FUNCTION_BLOCK CiA_DS402Controlword_Lenze EXTENDS CiA_DS402Controlword
VAR_INPUT
	ReleaseBrake			: BOOL; //Manufacturere specific Bit 14 
END_VAR
VAR_OUTPUT
END_VAR
VAR
END_VAR

;

METHOD PUBLIC createControlword : BOOL
VAR_INPUT
	StatusState												: eCiA_DS402_STATUS_STATE;
END_VAR
VAR_IN_OUT
	Controlword												:	UINT;
END_VAR
	
	createControlword											:= SUPER^.createControlword(StatusState,Controlword);;
	Controlword.14												:= ReleaseBrake;	
	
	

(*****************************************************************************)
END_METHOD

END_FUNCTION_BLOCK

(* stored: Version 1.1.0.1, ProductVersion 3.1.4024.13
   POU CiA_DS402Controlword_Lenze: Id {8f5f011b-553f-44e1-a91b-77b2decd4123}, SpecialFunc None
   Method createControlword: Id {b954e133-1a8a-44f1-88e1-a55de35a506f} *)
